VAR_GLOBAL 
  sPLC_TO_PC   			AT%MW400  :DUT_PCReceive;
  sPLC_From_PC  		AT%MW0    :DUT_PCSend;
  sCamera_TO_Plc 		AT%MW100  :DUT_CameraSend;
	sCamera_From_Plc	AT%MW150	:DUT_CameraReceive;
  sModbus_200SMART :DUT_200SMART;
END_VAR

(* stored: Version 1.1.0.1, ProductVersion 3.1.4024.9
   GVL GVL_PC: Id {dc3939c5-e481-4168-9b1e-3e5db0363608} *)
